(* CoDeSys 2.3 export: MAP_INT.EXP *)

(* POU FB_LIBRARY/MAP_INT, ST *)
FUNCTION MAP_INT : INT
(*
Author: Nikshitha S
Date: 10-08-2023
Description: This particular function works on inputs and outputs both with INTEGER datatype. Thus consuming less memory.
*)
VAR_INPUT
	IN: INT;
	IN_MIN:INT;
	IN_MAX : INT;
	OUT_MIN:INT;
	OUT_MAX:INT;
END_VAR

VAR
	ERROR: BOOL;
	FINAL_MAP: INT;
	INPUT_RANGE: INT;
	OUTPUT_RANGE: INT;
END_VAR
ERROR := (IN_MAX-IN_MIN=0) OR (IN<IN_MIN) OR (IN>IN_MAX);

INPUT_RANGE := IN_MAX-IN_MIN;
OUTPUT_RANGE := OUT_MAX-OUT_MIN;

MAP_INT:= ((IN-IN_MIN)*OUTPUT_RANGE) / INPUT_RANGE + OUT_MIN;


IF ERROR AND (IN<IN_MIN)THEN
MAP_INT:=OUT_MIN;
END_IF

IF ERROR AND (IN>IN_MAX)THEN
MAP_INT:=OUT_MAX;
END_IF
END_FUNCTION
